// TIA Portal V18 export
FUNCTION "_coordinate_database_manager_main" : Void   // FC14, FBD
{ S7_Optimized_Access := 'TRUE' }
VERSION : 0.1
// stored: AutoNumber true, IsIECCheckEnabled false, SetENOAutomatically false, UDAEnableTagReadback false
BEGIN

REGION Network 1
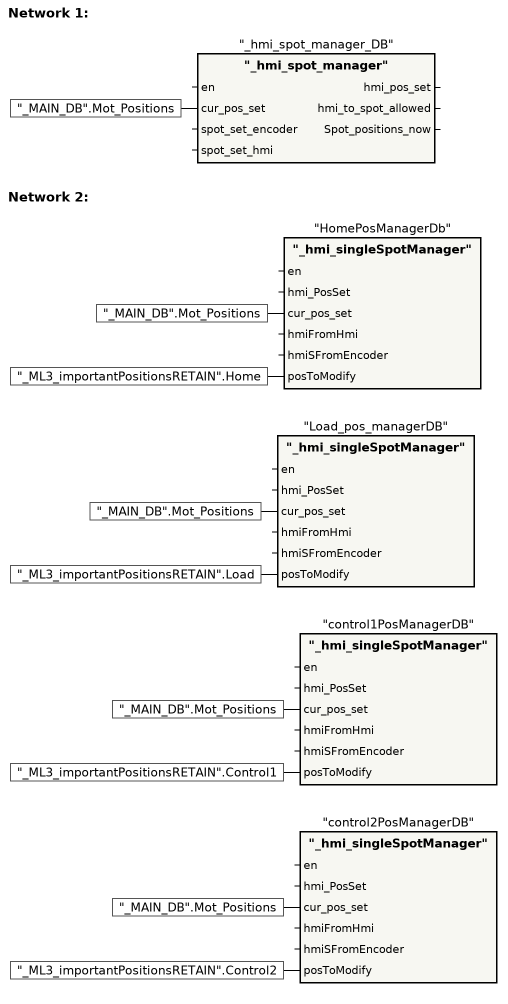
   "_hmi_spot_manager_DB"(cur_pos_set := "_MAIN_DB".Mot_Positions);   // "_hmi_spot_manager"
END_REGION

REGION Network 2
   "HomePosManagerDb"(cur_pos_set := "_MAIN_DB".Mot_Positions,   // "_hmi_singleSpotManager"
                      posToModify := "_ML3_importantPositionsRETAIN".Home);
   "Load_pos_managerDB"(cur_pos_set := "_MAIN_DB".Mot_Positions,   // "_hmi_singleSpotManager"
                        posToModify := "_ML3_importantPositionsRETAIN".Load);
   "control1PosManagerDB"(cur_pos_set := "_MAIN_DB".Mot_Positions,   // "_hmi_singleSpotManager"
                          posToModify := "_ML3_importantPositionsRETAIN".Control1);
   "control2PosManagerDB"(cur_pos_set := "_MAIN_DB".Mot_Positions,   // "_hmi_singleSpotManager"
                          posToModify := "_ML3_importantPositionsRETAIN".Control2);
END_REGION
END_FUNCTION
